SUBAPPLICATION Ventilsteuerung_Uebung_015 (* Object Pointer umschalten *)
  (* Standard: 61499-2 *)
  (* Version 1.0, 2023-10-23, franz *)
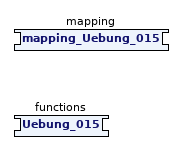
  SUBAPPS
    mapping : mapping_Uebung_015;
    functions : Uebung_015;
  END_SUBAPPS
END_SUBAPPLICATION
